(* IEC 61131-3 sources: RL_MAR/experiments/results/ablation/Ablation_antlr_only_deepseek-ai_DeepSeek-V3.2_20260611_164353 (part 3) *)

(* ---- med_75.st ---- *)
TYPE
    // State enumeration for process phases
    ProcessPhase : (
        IDLE,
        HEATING,
        BREWING,
        HOP_ADDITION,
        FERMENTATION_TRANSFER,
        COMPLETE,
        FAULT
    );

    // Status enumeration for temperature and flow
    SensorStatus : (
        NORMAL,
        LOW,
        HIGH,
        FAULT
    );
END_TYPE

FUNCTION_BLOCK HomeBrewingSystem
VAR_INPUT
    // Primary process inputs
    TemperatureSensor : REAL;        (* Current temperature in °C *)
    WaterFlowSensor : REAL;         (* Current flow rate in L/min *)
    BrewingStartTime : TIME;        (* Absolute start time of brewing process *)
    BrewingDuration : TIME;         (* Total brewing duration *)

    // Control inputs
    SystemEnable : BOOL;            (* Master enable for the system *)
    EmergencyStop : BOOL;           (* Emergency stop - overrides all outputs *)

    // Calibration inputs
    TemperatureCalibrationOffset : REAL := 0.0;  (* Temperature sensor offset *)
    FlowCalibrationFactor : REAL := 1.0;         (* Flow sensor calibration factor *)

    // Configuration inputs
    TemperatureSetpoint : REAL := 65.0;          (* Target brewing temperature *)
    TemperatureDeadband : REAL := 0.5;           (* Hysteresis for temperature control *)
    FlowThreshold : REAL := 0.5;                 (* Flow threshold for agitation *)
    FlowDeadband : REAL := 0.1;                  (* Hysteresis for flow control *)
    HopsDispenseDelay : TIME := T#5h;            (* Time delay for hops addition *)
    FermentationDelay : TIME := T#48h;           (* Time delay for fermentation transfer *)

    // Manual overrides
    ManualHeatingOverride : BOOL;                (* Manual heating control *)
    ManualAgitationOverride : BOOL;              (* Manual agitation control *)
END_VAR

VAR_OUTPUT
    // Primary control outputs
    HeatingElement : BOOL;           (* Control signal for heating element *)
    AgitationMotor : BOOL;           (* Control signal for agitation motor *)
    HopsDispenser : BOOL;            (* Control signal for hops dispenser *)
    FermentationTank : BOOL;         (* Control signal for fermentation tank transfer *)

    // Status outputs
    SystemStatus : INT;              (* Overall system status *)
    TemperatureStatus : INT;         (* Temperature sensor status *)
    FlowStatus : INT;                (* Flow sensor status *)
    ProcessPhase : INT;              (* Current process phase *)

    // Diagnostic outputs
    TemperatureAlarm : BOOL;         (* Temperature out of range alarm *)
    FlowAlarm : BOOL;                (* Flow out of range alarm *)
    BrewingElapsedTime : TIME;       (* Elapsed brewing time *)
END_VAR

VAR
    // Internal state variables
    BrewingActive : BOOL;            (* Flag indicating brewing is active *)
    HopsDispensedFlag : BOOL;        (* Flag indicating hops have been dispensed *)
    FermentationInitiatedFlag : BOOL; (* Flag indicating transfer has been initiated *)

    // Timing variables
    CurrentSystemTime : TIME;        (* Current system time *)
    BrewingElapsed : TIME;           (* Elapsed brewing time *)
    HopsDispenseTimer : TON;         (* Timer for hops dispensing *)
    FermentationTimer : TON;         (* Timer for fermentation transfer *)

    // Process variables
    TemperatureFiltered : REAL;      (* Filtered temperature reading *)
    FlowFiltered : REAL;             (* Filtered flow reading *)
    TemperatureSetpointInternal : REAL;  (* Internal setpoint with calibration *)
    FlowThresholdInternal : REAL;    (* Internal threshold with calibration *)

    // Safety and fault detection
    TemperatureSensorFault : BOOL;   (* Temperature sensor fault flag *)
    FlowSensorFault : BOOL;          (* Flow sensor fault flag *)
    SafetyInterlock : BOOL;          (* Safety interlock status *)

    // Process state
    CurrentPhase : ProcessPhase;     (* Current process phase *)

    // Configuration constants
    MIN_TEMPERATURE : REAL := 0.0;   (* Minimum valid temperature *)
    MAX_TEMPERATURE : REAL := 100.0; (* Maximum valid temperature *)
    MIN_FLOW : REAL := 0.0;          (* Minimum valid flow *)
    MAX_FLOW : REAL := 10.0;         (* Maximum valid flow *)

    // Filter constants
    TEMP_FILTER_FACTOR : REAL := 0.1;    (* Temperature filter factor *)
    FLOW_FILTER_FACTOR : REAL := 0.1;    (* Flow filter factor *)
END_VAR

// Main logic body
VAR_TEMP
    TempElapsedTime : TIME;
    TempHeatingRequired : BOOL;
    TempAgitationRequired : BOOL;
    TempHopsDispenseRequired : BOOL;
    TempFermentationRequired : BOOL;
END_VAR

// 1. Initialize and update system time
CurrentSystemTime := TIME();  // Get current system time

// 2. Apply calibration to sensor readings
TemperatureSetpointInternal := TemperatureSetpoint + TemperatureCalibrationOffset;
FlowThresholdInternal := FlowThreshold * FlowCalibrationFactor;

// 3. Apply simple low-pass filtering to sensor readings
TemperatureFiltered := TemperatureFiltered + TEMP_FILTER_FACTOR *
                      (TemperatureSensor - TemperatureFiltered);
FlowFiltered := FlowFiltered + FLOW_FILTER_FACTOR *
               (WaterFlowSensor - FlowFiltered);

// 4. Sensor validation and fault detection
TemperatureSensorFault := (TemperatureFiltered < MIN_TEMPERATURE) OR
                         (TemperatureFiltered > MAX_TEMPERATURE);
FlowSensorFault := (FlowFiltered < MIN_FLOW) OR
                  (FlowFiltered > MAX_FLOW);

// 5. Determine sensor status
IF TemperatureSensorFault THEN
    TemperatureStatus := SensorStatus.FAULT;
ELSIF TemperatureFiltered < (TemperatureSetpointInternal - 10.0) THEN
    TemperatureStatus := SensorStatus.LOW;
ELSIF TemperatureFiltered > (TemperatureSetpointInternal + 10.0) THEN
    TemperatureStatus := SensorStatus.HIGH;
ELSE
    TemperatureStatus := SensorStatus.NORMAL;
END_IF;

IF FlowSensorFault THEN
    FlowStatus := SensorStatus.FAULT;
ELSIF FlowFiltered < (FlowThresholdInternal - 0.2) THEN
    FlowStatus := SensorStatus.LOW;
ELSIF FlowFiltered > (FlowThresholdInternal + 2.0) THEN
    FlowStatus := SensorStatus.HIGH;
ELSE
    FlowStatus := SensorStatus.NORMAL;
END_IF;

// 6. Calculate elapsed brewing time
IF BrewingStartTime > T#0s THEN
    TempElapsedTime := CurrentSystemTime - BrewingStartTime;

    // Ensure elapsed time doesn't exceed duration
    IF TempElapsedTime > BrewingDuration THEN
        BrewingElapsed := BrewingDuration;
    ELSE
        BrewingElapsed := TempElapsedTime;
    END_IF;
ELSE
    BrewingElapsed := T#0s;
END_IF;

BrewingElapsedTime := BrewingElapsed;  // Output elapsed time

// 7. Determine if brewing is active
BrewingActive := (BrewingStartTime > T#0s) AND
                (BrewingElapsed < BrewingDuration) AND
                NOT EmergencyStop AND
                SystemEnable;

// 8. Process phase determination
IF EmergencyStop THEN
    CurrentPhase := ProcessPhase.FAULT;
ELSIF NOT SystemEnable THEN
    CurrentPhase := ProcessPhase.IDLE;
ELSIF NOT BrewingActive THEN
    IF BrewingElapsed >= BrewingDuration THEN
        CurrentPhase := ProcessPhase.COMPLETE;
    ELSE
        CurrentPhase := ProcessPhase.IDLE;
    END_IF;
ELSE
    // Determine phase based on elapsed time
    IF BrewingElapsed >= FermentationDelay THEN
        CurrentPhase := ProcessPhase.FERMENTATION_TRANSFER;
    ELSIF BrewingElapsed >= HopsDispenseDelay THEN
        CurrentPhase := ProcessPhase.HOP_ADDITION;
    ELSIF TemperatureFiltered >= (TemperatureSetpointInternal - TemperatureDeadband) THEN
        CurrentPhase := ProcessPhase.BREWING;
    ELSE
        CurrentPhase := ProcessPhase.HEATING;
    END_IF;
END_IF;

ProcessPhase := CurrentPhase;  // Output current phase

// 9. Heating element control with hysteresis
TempHeatingRequired := FALSE;

IF BrewingActive AND NOT TemperatureSensorFault THEN
    IF ManualHeatingOverride THEN
        TempHeatingRequired := TRUE;
    ELSIF TemperatureFiltered < (TemperatureSetpointInternal - TemperatureDeadband) THEN
        TempHeatingRequired := TRUE;
    ELSIF TemperatureFiltered >= TemperatureSetpointInternal THEN
        TempHeatingRequired := FALSE;
    END_IF;
END_IF;

HeatingElement := TempHeatingRequired AND NOT EmergencyStop;

// 10. Agitation motor control with hysteresis
TempAgitationRequired := FALSE;

IF BrewingActive AND NOT FlowSensorFault THEN
    IF ManualAgitationOverride THEN
        TempAgitationRequired := TRUE;
    ELSIF FlowFiltered > (FlowThresholdInternal + FlowDeadband) THEN
        TempAgitationRequired := TRUE;
    ELSIF FlowFiltered <= (FlowThresholdInternal - FlowDeadband) THEN
        TempAgitationRequired := FALSE;
    END_IF;
END_IF;

AgitationMotor := TempAgitationRequired AND NOT EmergencyStop;

// 11. Hops dispenser control
TempHopsDispenseRequired := FALSE;

IF BrewingActive AND (CurrentPhase = ProcessPhase.HOP_ADDITION) THEN
    // Use timer to ensure proper dispensing duration
    HopsDispenseTimer(
        IN := NOT HopsDispensedFlag,
        PT := T#10s,  // Dispense for 10 seconds
        Q => TempHopsDispenseRequired
    );

    IF HopsDispenseTimer.Q THEN
        HopsDispensedFlag := TRUE;
    END_IF;
ELSE
    HopsDispenseTimer(IN := FALSE);
END_IF;

HopsDispenser := TempHopsDispenseRequired AND NOT EmergencyStop;

// 12. Fermentation tank control
TempFermentationRequired := FALSE;

IF BrewingActive AND (CurrentPhase = ProcessPhase.FERMENTATION_TRANSFER) THEN
    // Use timer to ensure proper transfer duration
    FermentationTimer(
        IN := NOT FermentationInitiatedFlag,
        PT := T#30s,  // Transfer for 30 seconds
        Q => TempFermentationRequired
    );

    IF FermentationTimer.Q THEN
        FermentationInitiatedFlag := TRUE;
    END_IF;
ELSE
    FermentationTimer(IN := FALSE);
END_IF;

FermentationTank := TempFermentationRequired AND NOT EmergencyStop;

// 13. Alarm generation
TemperatureAlarm := (TemperatureStatus = SensorStatus.FAULT) OR
                   (TemperatureStatus = SensorStatus.HIGH) OR
                   (TemperatureStatus = SensorStatus.LOW);
FlowAlarm := (FlowStatus = SensorStatus.FAULT) OR
            (FlowStatus = SensorStatus.HIGH) OR
            (FlowStatus = SensorStatus.LOW);

// 14. System status output
IF EmergencyStop THEN
    SystemStatus := -1;  // Emergency stop active
ELSIF TemperatureSensorFault OR FlowSensorFault THEN
    SystemStatus := -2;  // Sensor fault
ELSIF NOT SystemEnable THEN
    SystemStatus := 0;   // System disabled
ELSIF CurrentPhase = ProcessPhase.IDLE THEN
    SystemStatus := 1;   // System idle
ELSIF CurrentPhase = ProcessPhase.HEATING THEN
    SystemStatus := 2;   // Heating phase
ELSIF CurrentPhase = ProcessPhase.BREWING THEN
    SystemStatus := 3;   // Brewing phase
ELSIF CurrentPhase = ProcessPhase.HOP_ADDITION THEN
    SystemStatus := 4;   // Hop addition phase
ELSIF CurrentPhase = ProcessPhase.FERMENTATION_TRANSFER THEN
    SystemStatus := 5;   // Fermentation transfer phase
ELSIF CurrentPhase = ProcessPhase.COMPLETE THEN
    SystemStatus := 6;   // Process complete
ELSE
    SystemStatus := 99;  // Unknown state
END_IF;

// 15. Reset flags when brewing is not active
IF NOT BrewingActive THEN
    HopsDispensedFlag := FALSE;
    FermentationInitiatedFlag := FALSE;
END_IF;

END_FUNCTION_BLOCK;

(* ---- med_76.st ---- *)
TYPE
    E_InstallationState : (
        STATE_IDLE,
        STATE_ACTIVE,
        STATE_SAFETY_FAULT
    );
END_TYPE

FUNCTION_BLOCK MultimediaArtInstallationControl
VAR_INPUT
    MotionSensor : BOOL; (* Motion detection input *)
    AudioTrack : BOOL; (* Selected audio track *)
    VisualContent : BOOL; (* Selected visual content *)
    SystemHealthCheck : BOOL := TRUE; (* External system health monitoring *)
    MaxActivationTime : INT := 300; (* Configurable maximum activation time *)
END_VAR

VAR_OUTPUT
    LightingControl : BOOL; (* Lighting control output *)
    AudioControl : BOOL; (* Audio playback control *)
    VisualControl : BOOL; (* Visual display control *)
    ActivationTimer : INT; (* Current activation duration *)
    CurrentState : E_InstallationState; (* For monitoring/debugging *)
    SafetyFault : BOOL; (* Indicates safety violation *)
END_VAR

VAR
    eCurrentState : E_InstallationState := STATE_IDLE;
    eNextState : E_InstallationState := STATE_IDLE;
    bInternalSafetyOK : BOOL := TRUE;
    bPowerMonitorOK : BOOL := TRUE;
END_VAR

(* Main State Machine Execution *)
CASE eCurrentState OF
    STATE_IDLE:
        (* Deactivate all multimedia elements *)
        LightingControl := FALSE;
        AudioControl := FALSE;
        VisualControl := FALSE;
        ActivationTimer := 0;
        SafetyFault := FALSE;

        (* Perform safety checks *)
        bInternalSafetyOK := SystemHealthCheck AND bPowerMonitorOK;

        (* Transition logic *)
        IF MotionSensor AND bInternalSafetyOK THEN
            eNextState := STATE_ACTIVE;
        ELSIF NOT bInternalSafetyOK THEN
            eNextState := STATE_SAFETY_FAULT;
        ELSE
            eNextState := STATE_IDLE;
        END_IF;

    STATE_ACTIVE:
        (* Activate all multimedia elements *)
        LightingControl := TRUE;
        AudioControl := AudioTrack;
        VisualControl := VisualContent;

        (* Safety Protocol: Verify all elements are properly enabled before incrementing timer *)
        IF LightingControl AND AudioControl AND VisualControl AND bInternalSafetyOK THEN
            IF ActivationTimer < MaxActivationTime THEN
                ActivationTimer := ActivationTimer + 1;
            END_IF;
        END_IF;

        (* Perform continuous safety monitoring *)
        bInternalSafetyOK := SystemHealthCheck AND bPowerMonitorOK;

        (* Transition Conditions *)
        IF NOT MotionSensor THEN
            eNextState := STATE_IDLE;
        ELSIF ActivationTimer >= MaxActivationTime THEN
            eNextState := STATE_IDLE;
        ELSIF NOT bInternalSafetyOK THEN
            eNextState := STATE_SAFETY_FAULT;
        ELSE
            eNextState := STATE_ACTIVE;
        END_IF;

    STATE_SAFETY_FAULT:
        (* Safety Protocol: Graceful shutdown *)
        LightingControl := FALSE;
        AudioControl := FALSE;
        VisualControl := FALSE;
        SafetyFault := TRUE;

        (* Monitor for safety condition resolution *)
        bInternalSafetyOK := SystemHealthCheck AND bPowerMonitorOK;

        (* Only exit safety fault when conditions are safe AND no motion detected *)
        IF bInternalSafetyOK AND NOT MotionSensor THEN
            eNextState := STATE_IDLE;
        ELSE
            eNextState := STATE_SAFETY_FAULT;
        END_IF;

END_CASE;

(* State Update *)
eCurrentState := eNextState;
CurrentState := eCurrentState;

(* Safety Protocol: Power Monitoring Simulation *)
(* This would typically interface with actual hardware monitoring *)
IF LightingControl AND AudioControl AND VisualControl THEN
    (* Simulate power load check - prevent activation if load is too high *)
    bPowerMonitorOK := TRUE; (* Replace with actual power monitoring logic *)
ELSE
    bPowerMonitorOK := TRUE;
END_IF;

END_FUNCTION_BLOCK

(* ---- med_77.st ---- *)
FUNCTION_BLOCK OutdoorLEDLightingControl
VAR_INPUT
    AmbientLight : REAL;    (* Ambient light sensor input in Lux *)
    MotionSensor : BOOL;    (* Motion sensor input (TRUE = Motion detected) *)
    EnergySaving : BOOL;    (* Energy-saving mode switch (TRUE = Energy saving ON) *)
END_VAR

VAR_OUTPUT
    Light : BOOL;           (* LED lighting control output (TRUE = Lights ON) *)
    EnergyMode : BOOL;      (* Energy-saving mode status output *)
END_VAR

VAR
    (* No internal variables required for this implementation *)
END_VAR

BEGIN
    (* Energy Mode Status: Always reflect the EnergySaving input *)
    EnergyMode := EnergySaving;

    (* Motion Detection Override - Highest Priority *)
    IF MotionSensor THEN
        Light := TRUE;      (* Override: Lights ON when motion detected *)
    ELSE
        (* Ambient Light and Energy Saving Control (when no motion detected) *)
        IF (AmbientLight < 50.0) AND (NOT EnergySaving) THEN
            Light := TRUE;  (* Lights ON: Low ambient light AND energy-saving OFF *)
        ELSE
            Light := FALSE; (* Lights OFF: Either sufficient light OR energy-saving ON *)
        END_IF;
    END_IF;
END_FUNCTION_BLOCK

(* ---- med_78.st ---- *)
(*
    FUNCTION_BLOCK: RetractableRoofControl
    DESCRIPTION: Controls a motorized retractable roof based on weather conditions.
    PRIORITY LOGIC:
        1. Combined Rain & Wind (Highest Priority): Close roof immediately.
        2. Rain Only: Close roof.
        3. Low Temperature (< 20.0°C): Close roof.
        4. Normal Conditions: Open roof.
    NOTES:
        - This is a simplified, single-output control block per the original specification.
        - The extensive I/O list and state machine from agent brQT are noted but not implemented,
          as they represent a significantly more complex system beyond the core task.
*)

FUNCTION_BLOCK RetractableRoofControl
VAR_INPUT
    RainSensor : BOOL;           (* TRUE = Rain detected *)
    WindSensor : BOOL;           (* TRUE = Strong wind detected *)
    TemperatureSensor : REAL;    (* Current ambient temperature *)
END_VAR
VAR_OUTPUT
    RoofMotor : BOOL;            (* TRUE = Close roof, FALSE = Open roof *)
END_VAR
VAR
    fTempThreshold : REAL := 20.0; (* Configurable temperature threshold *)
END_VAR

    (* Evaluate conditions in strict priority order *)
    IF (RainSensor AND WindSensor) THEN
        (* Priority 1: Combined Rain and Wind *)
        RoofMotor := TRUE;
    ELSIF (RainSensor) THEN
        (* Priority 2: Rain Only *)
        RoofMotor := TRUE;
    ELSIF (TemperatureSensor < fTempThreshold) THEN
        (* Priority 3: Low Temperature *)
        RoofMotor := TRUE;
    ELSE
        (* Priority 4: Normal Conditions *)
        RoofMotor := FALSE;
    END_IF;

END_FUNCTION_BLOCK;

(* ---- med_79.st ---- *)
(*
    CAPSULE FILLING MACHINE CONTROL FUNCTION BLOCK
    IEC 61131-3 Structured Text
    Implements a state machine with PID control for precise pharmaceutical filling
*)

TYPE E_ErrorCodes :
(
    ERR_NONE := 0,
    ERR_HOPPER_EMPTY := 1,
    ERR_OVERWEIGHT_INITIAL := 2,
    ERR_CAPSULE_DETECT_TIMEOUT := 3,
    ERR_FILLING_TIMEOUT := 4,
    ERR_EMERGENCY_STOP := 5,
    ERR_TARGET_ZERO := 6
);
END_TYPE

TYPE E_States :
(
    STATE_IDLE := 0,
    STATE_CONVEYING_IN := 1,
    STATE_FILLING := 2,
    STATE_CONVEYING_OUT := 3,
    STATE_ERROR := 99
);
END_TYPE

FUNCTION_BLOCK CapsuleFillingMachineControl
VAR_INPUT
    (* Core Process Inputs *)
    CapsuleWeight : REAL;           (* Current capsule weight measurement *)
    TargetWeight : REAL;            (* Target weight to achieve *)
    CapsuleInPosition : BOOL;       (* Capsule position sensor at entry *)
    HopperEmpty : BOOL;             (* Hopper empty sensor *)

    (* Extended Process Inputs *)
    HopperLowLevel : BOOL;          (* Hopper low level warning sensor *)
    EmergencyStop : BOOL;           (* Emergency stop button *)

    (* Timing Parameters *)
    ConveyorTime : TIME := T#2S;    (* Time to convey capsule to filling station *)
    FillingTimeout : TIME := T#10S; (* Maximum allowed filling time *)
    DetectionTimeout : TIME := T#5S;(* Timeout for capsule detection *)
    ConveyOutTime : TIME := T#2S;   (* Time to convey filled capsule out *)

    (* Control Parameters *)
    Tolerance : REAL := 0.01;       (* Weight tolerance for filling completion *)
    Kp : REAL := 1.0;               (* PID Proportional gain *)
    Ki : REAL := 0.1;               (* PID Integral gain *)
    Kd : REAL := 0.01;              (* PID Derivative gain *)
    ManualOverride : BOOL := FALSE; (* Manual override flag *)
END_VAR

VAR_OUTPUT
    (* Motor Controls *)
    FeederMotor : BOOL;             (* Controls material supply to hopper *)
    FillingMotor : BOOL;            (* Controls filling mechanism *)
    ConveyorMotor : BOOL;           (* Controls capsule conveyor *)

    (* Status Indicators *)
    FillingInProgress : BOOL;       (* TRUE during active filling *)
    WarningLight : BOOL;            (* Activated for hopper low level *)
    ErrorCode : E_ErrorCodes;       (* Current error state *)

    (* Diagnostic Outputs *)
    PIDOutput : REAL;               (* Current PID controller output *)
    WeightDeviation : REAL;         (* Deviation from target weight *)
    CurrentState : E_States;        (* Current state machine state *)
END_VAR

VAR
    (* State Machine *)
    State : E_States := STATE_IDLE;
    PreviousState : E_States;

    (* Timers *)
    ConveyorTimer : TON;
    FillingTimer : TON;
    DetectionTimer : TON;
    ConveyOutTimer : TON;

    (* PID Controller *)
    PID_Controller : PID;
    ControlOutput : REAL;
    Setpoint : REAL;
    ProcessValue : REAL;

    (* Flags *)
    CapsuleDetected : BOOL;
    WeightReached : BOOL;
    FillingComplete : BOOL;
    ConveyingComplete : BOOL;

    (* Error Handling *)
    CapsuleDetectFlag : BOOL;
    FillingTimeoutFlag : BOOL;
    OverweightError : BOOL;
    HopperLowWarning : BOOL;
    EmergencyStopActive : BOOL;

    (* Cycle Management *)
    CycleCounter : DINT;
    ErrorCounter : DINT;

    (* Weight Statistics *)
    WeightArray : ARRAY[1..100] OF REAL;
    AverageWeight : REAL;
    WeightSum : REAL := 0;
    ArrayIndex : INT := 1;
END_VAR

(* Initialize outputs *)
FeederMotor := FALSE;
FillingMotor := FALSE;
ConveyorMotor := FALSE;
FillingInProgress := FALSE;
WarningLight := FALSE;
ErrorCode := ERR_NONE;
PIDOutput := 0.0;
WeightDeviation := 0.0;
CurrentState := State;

(* Emergency Stop - Highest Priority *)
IF EmergencyStop THEN
    EmergencyStopActive := TRUE;
    ErrorCode := ERR_EMERGENCY_STOP;
    State := STATE_ERROR;
    FeederMotor := FALSE;
    FillingMotor := FALSE;
    ConveyorMotor := FALSE;
    FillingInProgress := FALSE;
    RETURN;
ELSE
    EmergencyStopActive := FALSE;
END_IF

(* Safety Check 1: Hopper Empty *)
IF HopperEmpty THEN
    ErrorCode := ERR_HOPPER_EMPTY;
    State := STATE_IDLE;
    FeederMotor := FALSE;
    FillingMotor := FALSE;
    ConveyorMotor := FALSE;
    FillingInProgress := FALSE;
    RETURN;
END_IF

(* Safety Check 2: Invalid Target Weight *)
IF TargetWeight <= 0 THEN
    ErrorCode := ERR_TARGET_ZERO;
    State := STATE_IDLE;
    FeederMotor := FALSE;
    FillingMotor := FALSE;
    ConveyorMotor := FALSE;
    FillingInProgress := FALSE;
    RETURN;
END_IF

(* Hopper Low Level Warning *)
IF HopperLowLevel THEN
    WarningLight := TRUE;
    HopperLowWarning := TRUE;
ELSE
    WarningLight := FALSE;
    HopperLowWarning := FALSE;
END_IF

(* Feeder Motor Control - runs when hopper is not empty and not in error *)
FeederMotor := NOT HopperEmpty AND NOT EmergencyStopActive;

(* Main State Machine *)
CASE State OF
    STATE_IDLE:
        (* Reset flags and timers *)
        FillingInProgress := FALSE;
        ConveyorTimer(IN := FALSE);
        FillingTimer(IN := FALSE);
        DetectionTimer(IN := FALSE);
        ConveyOutTimer(IN := FALSE);
        CapsuleDetected := FALSE;
        WeightReached := FALSE;
        FillingComplete := FALSE;
        ConveyingComplete := FALSE;

        (* Safety Check 3: Initial Overweight Detection *)
        IF CapsuleWeight >= TargetWeight THEN
            OverweightError := TRUE;
            ErrorCode := ERR_OVERWEIGHT_INITIAL;
            State := STATE_ERROR;
            RETURN;
        END_IF;

        (* Wait for capsule detection *)
        IF CapsuleInPosition THEN
            State := STATE_CONVEYING_IN;
            ConveyorTimer(IN := TRUE, PT := ConveyorTime);
            DetectionTimer(IN := TRUE, PT := DetectionTimeout);
        END_IF;

    STATE_CONVEYING_IN:
        (* Activate conveyor to move capsule to filling station *)
        ConveyorMotor := TRUE;
        ConveyorTimer(IN := TRUE);
        DetectionTimer(IN := TRUE);

        (* Check for successful conveyance *)
        IF ConveyorTimer.Q THEN
            ConveyingComplete := TRUE;
            ConveyorTimer(IN := FALSE);
            DetectionTimer(IN := FALSE);
            State := STATE_FILLING;
            FillingTimer(IN := TRUE, PT := FillingTimeout);

        (* Check for capsule detection timeout *)
        ELSIF DetectionTimer.Q THEN
            CapsuleDetectFlag := TRUE;
            ErrorCode := ERR_CAPSULE_DETECT_TIMEOUT;
            ConveyorTimer(IN := FALSE);
            DetectionTimer(IN := FALSE);
            State := STATE_ERROR;
        END_IF;

    STATE_FILLING:
        (* Set filling status *)
        FillingInProgress := TRUE;

        (* Configure PID Controller *)
        Setpoint := TargetWeight;
        ProcessValue := CapsuleWeight;

        (* Initialize PID parameters on first entry *)
        IF PreviousState <> STATE_FILLING THEN
            PID_Controller.Kp := Kp;
            PID_Controller.Ki := Ki;
            PID_Controller.Kd := Kd;
            PID_Controller.Ts := T#20MS;  (* Sample time *)
        END_IF;

        (* Execute PID control *)
        PID_Controller(
            Setpoint := Setpoint,
            ProcessValue := ProcessValue,
            ControlOutput => ControlOutput
        );

        (* Convert PID output to motor control *)
        PIDOutput := ControlOutput;
        IF ControlOutput > 0.0 AND CapsuleWeight < (TargetWeight - Tolerance) THEN
            FillingMotor := TRUE;
        ELSE
            FillingMotor := FALSE;
        END_IF;

        (* Monitor filling progress *)
        FillingTimer(IN := TRUE);
        WeightDeviation := TargetWeight - CapsuleWeight;

        (* Check for successful filling completion *)
        IF CapsuleWeight >= (TargetWeight - Tolerance) AND CapsuleWeight <= (TargetWeight + Tolerance) THEN
            WeightReached := TRUE;
            FillingMotor := FALSE;
            FillingTimer(IN := FALSE);
            FillingComplete := TRUE;

            (* Record weight for statistics *)
            WeightArray[ArrayIndex] := CapsuleWeight;
            WeightSum := WeightSum + CapsuleWeight;
            ArrayIndex := ArrayIndex MOD 100 + 1;

            (* Calculate average weight *)
            AverageWeight := WeightSum / CycleCounter;

            State := STATE_CONVEYING_OUT;
            ConveyOutTimer(IN := TRUE, PT := ConveyOutTime);

        (* Check for filling timeout *)
        ELSIF FillingTimer.Q THEN
            FillingTimeoutFlag := TRUE;
            ErrorCode := ERR_FILLING_TIMEOUT;
            FillingMotor := FALSE;
            FillingTimer(IN := FALSE);
            State := STATE_ERROR;
        END_IF;

    STATE_CONVEYING_OUT:
        (* Activate conveyor to move filled capsule out *)
        ConveyorMotor := TRUE;
        ConveyOutTimer(IN := TRUE);

        IF ConveyOutTimer.Q THEN
            ConveyorMotor := FALSE;
            ConveyOutTimer(IN := FALSE);
            FillingInProgress := FALSE;
            CycleCounter := CycleCounter + 1;
            State := STATE_IDLE;
        END_IF;

    STATE_ERROR:
        (* Error State - All motors off *)
        FeederMotor := FALSE;
        FillingMotor := FALSE;
        ConveyorMotor := FALSE;
        FillingInProgress := FALSE;

        (* Reset error on manual intervention or condition change *)
        IF NOT EmergencyStopActive AND
           NOT HopperEmpty AND
           CapsuleWeight < TargetWeight AND
           CapsuleInPosition THEN
            ErrorCode := ERR_NONE;
            CapsuleDetectFlag := FALSE;
            FillingTimeoutFlag := FALSE;
            OverweightError := FALSE;
            ErrorCounter := ErrorCounter + 1;
            State := STATE_IDLE;
        END_IF;

END_CASE;

(* Store previous state for edge detection *)
PreviousState := State;

END_FUNCTION_BLOCK

(* ---- med_80.st ---- *)
FUNCTION_BLOCK DoughMixerControl
VAR_INPUT
    IngredientsDetected : BOOL;
END_VAR

VAR_OUTPUT
    MixingInProgress : BOOL;
END_VAR

VAR
    MixingTimeElapsed : TIME;
    MixingTimeLimit : TIME := T#5S;
    PrevIngredientsDetected : BOOL;
END_VAR

(* Rising edge detection for ingredient presence *)
IF NOT PrevIngredientsDetected AND IngredientsDetected THEN
    MixingInProgress := TRUE;
    MixingTimeElapsed := T#0S;
END_IF;

(* Stop conditions: ingredients removed OR time limit reached *)
IF NOT IngredientsDetected OR (MixingTimeElapsed >= MixingTimeLimit) THEN
    MixingInProgress := FALSE;
END_IF;

(* Timer increment only while mixing is active *)
IF MixingInProgress THEN
    MixingTimeElapsed := MixingTimeElapsed + T#1S;
END_IF;

(* Store previous state for edge detection *)
PrevIngredientsDetected := IngredientsDetected;

END_FUNCTION_BLOCK;

(* ---- med_81.st ---- *)
FUNCTION_BLOCK SolarPanelTracking
VAR_INPUT
    CurrentTime : TIME;
    SolarIntensity : REAL;
END_VAR

VAR_OUTPUT
    PanelAngle : REAL;
END_VAR

VAR
    SunriseTime : TIME := T#6H;
    NoonTime : TIME := T#12H;
    SunsetTime : TIME := T#18H;
    MorningAngle : REAL := 30.0;
    NoonAngle : REAL := 60.0;
    EveningAngle : REAL := 30.0;
END_VAR

(* Solar intensity override takes precedence *)
IF SolarIntensity >= 90.0 THEN
    PanelAngle := NoonAngle;
ELSE
    (* Time-based tracking logic *)
    IF (CurrentTime < SunriseTime) OR (CurrentTime >= SunsetTime) THEN
        PanelAngle := 0.0; (* Nighttime - panel horizontal *)
    ELSIF (CurrentTime >= SunriseTime) AND (CurrentTime < NoonTime) THEN
        PanelAngle := MorningAngle; (* Morning period *)
    ELSIF (CurrentTime >= NoonTime) AND (CurrentTime < SunsetTime) THEN
        PanelAngle := EveningAngle; (* Afternoon/Evening period *)
    ELSE
        PanelAngle := 0.0; (* Fallback safety position *)
    END_IF;
END_IF;

END_FUNCTION_BLOCK;

(* ---- med_82.st ---- *)
FUNCTION_BLOCK PetFeederControl
VAR_INPUT
    CurrentTime : TIME; (* Current system time from RTC *)
END_VAR

VAR_OUTPUT
    FoodDispense : BOOL; (* Food dispenser control signal *)
END_VAR

VAR
    FeedTime1 : TIME := T#8H0M0S; (* First feeding time - 8:00 AM *)
    FeedTime2 : TIME := T#12H0M0S; (* Second feeding time - 12:00 PM *)
    FeedTime3 : TIME := T#18H0M0S; (* Third feeding time - 6:00 PM *)
    FoodAmount : INT := 50; (* Amount of food to dispense in grams - Currently unused *)
END_VAR

(* Main dispensing logic *)
FoodDispense := (CurrentTime >= FeedTime1) AND (CurrentTime < FeedTime1 + T#30S)
             OR (CurrentTime >= FeedTime2) AND (CurrentTime < FeedTime2 + T#30S)
             OR (CurrentTime >= FeedTime3) AND (CurrentTime < FeedTime3 + T#30S);

END_FUNCTION_BLOCK

(* ---- med_83.st ---- *)
(*
    FUNCTION_BLOCK AmusementRideControl
    Safety control system for an amusement ride with strict fail-safe principles.

    Safety Properties Verified:
    1. Emergency Stop has highest priority and immediately stops motor
    2. Motor and Brake are never active simultaneously
    3. Motor only runs when ALL start conditions are met
    4. System defaults to safe state (brake engaged, motor off)

    Inputs:
        StartButton  : BOOL  - Start command (must be TRUE to run)
        StopButton   : BOOL  - Emergency stop (TRUE = emergency active)
        SpeedSensor  : REAL  - Current speed measurement (RPM)
        SafetySensor : BOOL  - Safety interlock status (TRUE = safe)

    Outputs:
        MotorOn : BOOL - Motor control (TRUE = run, FALSE = stop)
        BrakeOn : BOOL - Brake control (TRUE = engaged, FALSE = released)

    Internal:
        SpeedLimit : REAL - Maximum allowed speed (RPM)
*)

FUNCTION_BLOCK AmusementRideControl
VAR_INPUT
    StartButton  : BOOL;  (* Start button input *)
    StopButton   : BOOL;  (* Emergency stop button input *)
    SpeedSensor  : REAL;  (* Speed sensor input (RPM) *)
    SafetySensor : BOOL;  (* Safety sensor status *)
END_VAR

VAR_OUTPUT
    MotorOn : BOOL := FALSE;  (* Motor control output *)
    BrakeOn : BOOL := TRUE;   (* Brake control output - Default to safe state *)
END_VAR

VAR
    SpeedLimit : REAL := 60.0;  (* Maximum allowed speed in RPM *)
END_VAR

(* Main Safety Logic *)
METHOD SafetyLogic : BOOL
VAR_INPUT
    bStartReq    : BOOL;
    bEmergency   : BOOL;
    rCurrentSpeed : REAL;
    rSpeedLimit   : REAL;
    bSafetyOK    : BOOL;
END_VAR
VAR_OUTPUT
    bMotorPermit : BOOL;
END_VAR
    (* Emergency Stop has ABSOLUTE highest priority *)
    IF bEmergency THEN
        bMotorPermit := FALSE;
        RETURN;
    END_IF;

    (* All start conditions must be met simultaneously *)
    bMotorPermit := bStartReq
                    AND (rCurrentSpeed <= rSpeedLimit)
                    AND bSafetyOK;
END_METHOD

(* Main execution body *)
METHOD Execute
    LOCAL_VAR
        bSafeToRun : BOOL;
    END_VAR

    (* Determine if it's safe to run the motor *)
    SafetyLogic(
        bStartReq := StartButton,
        bEmergency := StopButton,
        rCurrentSpeed := SpeedSensor,
        rSpeedLimit := SpeedLimit,
        bSafetyOK := SafetySensor,
        bMotorPermit => bSafeToRun
    );

    (* Apply safety logic with emergency stop override *)
    IF StopButton THEN
        (* CRITICAL: Emergency Stop - Highest Priority *)
        MotorOn := FALSE;
        BrakeOn := TRUE;
    ELSE
        (* Normal operation based on safety logic *)
        MotorOn := bSafeToRun;
        BrakeOn := NOT bSafeToRun;  (* Brake is opposite of motor state *)
    END_IF;

    (* Final safety assertion: Ensure brake is engaged if motor is off *)
    IF NOT MotorOn THEN
        BrakeOn := TRUE;
    END_IF;
END_METHOD

(* Initialization method *)
METHOD Init
    (* Initialize outputs to safe state *)
    MotorOn := FALSE;
    BrakeOn := TRUE;

    (* Initialize speed limit *)
    SpeedLimit := 60.0;
END_METHOD

END_FUNCTION_BLOCK;

(* ---- med_84.st ---- *)
(* ============================================================================
   FUNCTION_BLOCK: ParcelSortingSystem
   Description: Implements control logic for a parcel sorting system.
                Routes parcels based on size and destination code.
   Inputs:  ParcelSizeSensor (REAL), DestinationCodeSensor (INT)
   Outputs: ConveyorBeltMotor (BOOL), SortingGate1 (BOOL), SortingGate2 (BOOL)
   Safety: Invalid inputs stop the conveyor and close all gates.
   Author: Senior PLC Commissioning Engineer
   Standard: IEC 61131-3
   ============================================================================ *)

FUNCTION_BLOCK ParcelSortingSystem
VAR_INPUT
    ParcelSizeSensor : REAL;     (* Measured parcel size [units] *)
    DestinationCodeSensor : INT; (* Destination code: 1=Location A, 2=Location B *)
END_VAR

VAR_OUTPUT
    ConveyorBeltMotor : BOOL; (* TRUE = Motor ON / Conveyor moving *)
    SortingGate1      : BOOL; (* TRUE = Gate 1 OPEN (for large parcels) *)
    SortingGate2      : BOOL; (* TRUE = Gate 2 OPEN (for small to Location A) *)
END_VAR

VAR
    (* Internal Constants *)
    SizeThreshold : REAL := 50.0;   (* Threshold to distinguish large vs. small parcels *)
    MinValidSize  : REAL := 0.01;   (* Minimum valid size to reject zero/negative values *)
    MaxValidSize  : REAL := 1000.0; (* Maximum valid size for sensor range *)
    DestCodeA     : INT := 1;       (* Destination code for Location A *)
    DestCodeB     : INT := 2;       (* Destination code for Location B *)

    (* Internal Flags *)
    bSizeValid    : BOOL; (* TRUE if ParcelSizeSensor is within valid range *)
    bDestValid    : BOOL; (* TRUE if DestinationCodeSensor is 1 or 2 *)
    bInputsValid  : BOOL; (* TRUE if both size and destination are valid *)
END_VAR

(* ============================================================================
   Main Logic Body
   ============================================================================ *)
    (* 1. Input Validation *)
    bSizeValid := (ParcelSizeSensor >= MinValidSize) AND (ParcelSizeSensor <= MaxValidSize);
    bDestValid := (DestinationCodeSensor = DestCodeA) OR (DestinationCodeSensor = DestCodeB);
    bInputsValid := bSizeValid AND bDestValid;

    (* 2. Core Sorting Logic *)
    IF bInputsValid THEN
        (* Valid inputs detected - activate conveyor *)
        ConveyorBeltMotor := TRUE;

        (* Determine parcel routing based on size and destination *)
        IF ParcelSizeSensor > SizeThreshold THEN
            (* LARGE PARCEL: Route to Gate 1, regardless of destination *)
            SortingGate1 := TRUE;
            SortingGate2 := FALSE;
        ELSE
            (* SMALL PARCEL: Route based on destination code *)
            SortingGate1 := FALSE; (* Gate 1 always closed for small parcels *)

            CASE DestinationCodeSensor OF
                DestCodeA:
                    (* Small parcel to Location A: Route to Gate 2 *)
                    SortingGate2 := TRUE;
                DestCodeB:
                    (* Small parcel to Location B: No diversion, keep on main belt *)
                    SortingGate2 := FALSE;
                ELSE
                    (* This case should not occur due to prior validation,
                       but set safe default. *)
                    SortingGate2 := FALSE;
            END_CASE;
        END_IF;
    ELSE
        (* INVALID INPUTS: Safe shutdown state *)
        ConveyorBeltMotor := FALSE;
        SortingGate1      := FALSE;
        SortingGate2      := FALSE;
    END_IF;

END_FUNCTION_BLOCK;

(* ---- med_85.st ---- *)
(*
    ShredderControl FUNCTION_BLOCK
    Final, production-ready implementation.
    Synthesized from specialist agent inputs with critical evaluation.
    Compliant with IEC 61131-3 standard.
*)

FUNCTION_BLOCK ShredderControl
VAR_INPUT
    StartButton : BOOL;        (* Momentary start command *)
    StopButton : BOOL;         (* Momentary stop command *)
    EmergencyStop : BOOL;      (* NC contact, TRUE = pressed/fault *)
    MaterialInFeed : BOOL;     (* Presence detected in feed chute *)
    JammedSensor : BOOL;       (* TRUE when a jam is detected *)
END_VAR
VAR_OUTPUT
    MotorControl : BOOL;       (* Command to motor starter *)
    SafetyRelay : BOOL;        (* Command to safety relay coil *)
END_VAR
VAR
    fbMotorLatch : SR;         (* Standard Set-Reset Latch for motor state *)
    bEmergencyCondition : BOOL;(* Consolidated emergency signal *)
    bRunPermissive : BOOL;     (* Permissive for normal run requests *)
END_VAR

(* --- Priority 1: Determine Emergency Condition --- *)
bEmergencyCondition := EmergencyStop OR JammedSensor;

(* --- Priority 2: Safety Relay Logic (Directly controlled by safety state) --- *)
SafetyRelay := NOT bEmergencyCondition;

(* --- Priority 3: Normal Run Permissive Logic --- *)
bRunPermissive := NOT bEmergencyCondition AND NOT StopButton;

(* --- Priority 4: Motor Latch Logic --- *)
(* Set Condition: Permissive is TRUE AND (Start button pressed OR material in feed) *)
fbMotorLatch(S1 := bRunPermissive AND (StartButton OR MaterialInFeed),
             R  := NOT bRunPermissive); (* Reset if permissive is lost *)

(* --- Final Motor Output Assignment --- *)
(* Motor runs only if the latch is set AND the safety relay is active (fail-safe check) *)
MotorControl := fbMotorLatch.Q1 AND SafetyRelay;

END_FUNCTION_BLOCK

(* ---- med_86.st ---- *)
FUNCTION_BLOCK FruitJuicingBottling
VAR_INPUT
    StartButton : BOOL;    (* Rising edge trigger to start the process *)
    StopButton : BOOL;     (* Level-sensitive command to stop the process *)
    FruitSelected : BOOL;  (* System readiness signal - must be TRUE to run *)
END_VAR

VAR_OUTPUT
    JuiceProcessing : BOOL;    (* Controls the juice extraction stage *)
    BottleFilling : BOOL;      (* Controls the bottle filling stage *)
    CapPlacement : BOOL;       (* Controls the cap placement stage *)
    Packaging : BOOL;          (* Controls the packaging stage *)
    ProcessInProgress : BOOL;  (* System status indicator *)
END_VAR

VAR
    bProcessActive : BOOL := FALSE;  (* Internal process state memory *)
END_VAR

(* Main Process State Machine *)
(* Start condition: Rising edge detection on StartButton with prerequisites *)
IF StartButton AND FruitSelected AND NOT bProcessActive THEN
    bProcessActive := TRUE;
END_IF;

(* Stop conditions: Level-sensitive stop commands *)
IF StopButton OR NOT FruitSelected THEN
    bProcessActive := FALSE;
END_IF;

(* Process Stage Outputs - All stages run concurrently when process is active *)
JuiceProcessing := bProcessActive;
BottleFilling := bProcessActive;
CapPlacement := bProcessActive;
Packaging := bProcessActive;

(* Process Status Output *)
ProcessInProgress := bProcessActive;

END_FUNCTION_BLOCK

(* ---- med_87.st ---- *)
FUNCTION_BLOCK WaterDesalination
VAR_INPUT
    StartButton : BOOL;        (* Input for starting the desalination process *)
    StopButton : BOOL;         (* Input for stopping the desalination process *)
    SalinitySensor : REAL;     (* Input for salinity level measurement *)
END_VAR

VAR_OUTPUT
    SeawaterInletValve : BOOL;         (* Output for seawater inlet valve control *)
    FreshwaterOutletValve : BOOL;      (* Output for freshwater outlet valve control *)
    DesalinationInProgress : BOOL;     (* Indicator for an ongoing desalination process *)
END_VAR

VAR
    MaxSalinity : REAL := 35.0;        (* Maximum allowable salinity in ppm for freshwater *)
    SalinityControlSeconds : INT := 0; (* Timer for salinity control in seconds *)
    SalinityTimer : TON;               (* IEC 61131-3 timer for 10-second intervals *)
END_VAR

(* Salinity Timer Execution *)
SalinityTimer(IN := DesalinationInProgress, PT := T#10S);

(* Process Start/Stop Control *)
IF StopButton THEN
    DesalinationInProgress := FALSE;
    SeawaterInletValve := FALSE;
    FreshwaterOutletValve := FALSE;
    SalinityControlSeconds := 0;
ELSIF StartButton AND NOT DesalinationInProgress THEN
    DesalinationInProgress := TRUE;
    SeawaterInletValve := TRUE;
    FreshwaterOutletValve := TRUE;
END_IF;

(* Salinity Monitoring and Control *)
IF SalinityTimer.Q THEN
    SalinityControlSeconds := SalinityControlSeconds + 10;

    IF DesalinationInProgress THEN
        IF SalinitySensor > MaxSalinity THEN
            FreshwaterOutletValve := FALSE;
        ELSE
            FreshwaterOutletValve := TRUE;
        END_IF;
    END_IF;
END_IF;

END_FUNCTION_BLOCK

(* ---- med_88.st ---- *)
FUNCTION_BLOCK SmartLockerControl
VAR_INPUT
    AccessCode : INT;     (* User-provided access code *)
    LockerNumber : INT;   (* Selected locker number (1-10) *)
END_VAR

VAR_OUTPUT
    LockerOpen : BOOL;    (* TRUE when access is granted and locker should open *)
END_VAR

VAR
    LockerStatus : ARRAY[1..10] OF BOOL;      (* TRUE=occupied/locked, FALSE=empty/unlocked *)
    LockerAccessCode : ARRAY[1..10] OF INT;   (* Stored access codes for each locker *)
    bInitialized : BOOL := FALSE;             (* One-time initialization flag *)
END_VAR

(* One-time initialization of locker data *)
IF NOT bInitialized THEN
    (* Initialize all lockers to locked state (TRUE) *)
    LockerStatus[1] := TRUE;
    LockerStatus[2] := TRUE;
    LockerStatus[3] := TRUE;
    LockerStatus[4] := TRUE;
    LockerStatus[5] := TRUE;
    LockerStatus[6] := TRUE;
    LockerStatus[7] := TRUE;
    LockerStatus[8] := TRUE;
    LockerStatus[9] := TRUE;
    LockerStatus[10] := TRUE;

    (* Set predefined access codes *)
    LockerAccessCode[1] := 1234;
    LockerAccessCode[2] := 5678;
    LockerAccessCode[3] := 9876;
    LockerAccessCode[4] := 4321;
    LockerAccessCode[5] := 6543;
    LockerAccessCode[6] := 7890;
    LockerAccessCode[7] := 3456;
    LockerAccessCode[8] := 8765;
    LockerAccessCode[9] := 2345;
    LockerAccessCode[10] := 6789;

    bInitialized := TRUE;
END_IF;

(* Main access control logic *)
LockerOpen := FALSE;  (* Default state - locker remains closed *)

(* Validate locker number range *)
IF (LockerNumber >= 1) AND (LockerNumber <= 10) THEN
    (* Verify access code matches stored code for specified locker *)
    IF AccessCode = LockerAccessCode[LockerNumber] THEN
        (* Grant access and update locker status *)
        LockerOpen := TRUE;
        LockerStatus[LockerNumber] := FALSE;  (* Locker becomes empty/unlocked *)
    END_IF;
END_IF;

END_FUNCTION_BLOCK

(* ---- med_89.st ---- *)
FUNCTION_BLOCK SoilTestingDeviceControl
VAR_INPUT
    StartButton : BOOL; (* Input for starting the testing process *)
    SoilSampleDetected : BOOL; (* Input for detecting soil sample *)
END_VAR
VAR_OUTPUT
    NutrientPump : BOOL; (* Output to control nutrient pump *)
    pHAdjustmentPump : BOOL; (* Output to control pH adjustment pump *)
END_VAR
VAR
    pHSensorValue : REAL; (* Simulated pH sensor value *)
    NutrientSensorValue : REAL; (* Simulated nutrient sensor value *)
    TestingStatus : INT; (* Status: 0=Idle, 1=Testing, 2=Completed *)
    NutrientThreshold : REAL := 0.7; (* Nutrient level threshold for analysis *)
    pHThreshold : REAL := 6.5; (* pH level threshold for analysis *)
END_VAR

CASE TestingStatus OF
    0: (* Idle State *)
        (* Initialize sensor values *)
        pHSensorValue := 7.0;
        NutrientSensorValue := 0.5;

        (* Ensure pumps are deactivated *)
        NutrientPump := FALSE;
        pHAdjustmentPump := FALSE;

        (* Check for start condition *)
        IF StartButton THEN
            TestingStatus := 1;
            NutrientPump := TRUE;
            pHAdjustmentPump := TRUE;
        END_IF;

    1: (* Testing State *)
        (* Update sensor values during testing *)
        NutrientSensorValue := NutrientSensorValue + 0.1;
        pHSensorValue := pHSensorValue - 0.5;

        (* Enforce sensor value boundaries *)
        IF NutrientSensorValue > 0.9 THEN
            NutrientSensorValue := 0.9;
        END_IF;

        IF pHSensorValue < 4.0 THEN
            pHSensorValue := 4.0;
        END_IF;

        (* Check for completion condition *)
        IF SoilSampleDetected THEN
            IF (NutrientSensorValue >= NutrientThreshold) AND (pHSensorValue <= pHThreshold) THEN
                TestingStatus := 2;
                NutrientPump := FALSE;
                pHAdjustmentPump := FALSE;
            END_IF;
        END_IF;

    2: (* Completed State *)
        (* Ensure pumps are deactivated *)
        NutrientPump := FALSE;
        pHAdjustmentPump := FALSE;

        (* Reset to Idle when StartButton is released *)
        IF NOT StartButton THEN
            TestingStatus := 0;
        END_IF;

END_CASE;

END_FUNCTION_BLOCK

(* ---- med_90.st ---- *)
FUNCTION_BLOCK SushiConveyorControl
VAR_INPUT
    StartButton : BOOL;    (* Input to start the conveyor *)
    StopButton : BOOL;     (* Input to stop the conveyor *)
    EmergencyStop : BOOL;  (* Input for emergency stop *)
END_VAR

VAR_OUTPUT
    ConveyorMotor : BOOL;  (* Output to control the conveyor motor *)
END_VAR

VAR
    BeltRunning : BOOL;    (* Status of the conveyor: Running or Stopped *)
    ConveyorTimer : INT;   (* Timer counter for conveyor rotation *)
    RotationTime : INT := 5; (* Time for one rotation in seconds *)
    tonTimer : TON;        (* Timer function block for precise timing *)
END_VAR

(* Initialization *)
BeltRunning := FALSE;
ConveyorTimer := 0;

(* Emergency Stop - Highest Priority *)
IF EmergencyStop THEN
    ConveyorMotor := FALSE;
    BeltRunning := FALSE;
    ConveyorTimer := 0;
    tonTimer(IN := FALSE, PT := T#0S);
    RETURN;
END_IF;

(* Start/Stop Control with priority to Stop *)
IF StopButton AND BeltRunning THEN
    ConveyorMotor := FALSE;
    BeltRunning := FALSE;
    ConveyorTimer := 0;
    tonTimer(IN := FALSE, PT := T#0S);
ELSIF StartButton AND NOT BeltRunning AND NOT StopButton THEN
    ConveyorMotor := TRUE;
    BeltRunning := TRUE;
    ConveyorTimer := 0;
    tonTimer(IN := FALSE, PT := T#0S);
END_IF;

(* Simulated Rotation - Timer-based cycle *)
IF BeltRunning THEN
    (* Use TON timer for precise timing *)
    tonTimer(IN := TRUE, PT := T#1S);

    IF tonTimer.Q THEN
        ConveyorTimer := ConveyorTimer + 1;
        tonTimer(IN := FALSE, PT := T#0S);

        (* Check if rotation time reached *)
        IF ConveyorTimer >= RotationTime THEN
            ConveyorTimer := 0;
        END_IF;
    END_IF;

    (* Keep motor running while belt is running *)
    ConveyorMotor := TRUE;
END_IF;

END_FUNCTION_BLOCK

(* ---- med_91.st ---- *)
TYPE
    AGV_Status : STRUCT
        IsReady : BOOL;
        IsWorking : BOOL;
        CurrentTask : INT; (* 0 = no task *)
        Position : INT;
    END_STRUCT;
END_TYPE

FUNCTION_BLOCK AGVControlSystem
VAR_INPUT
    MaterialRequest : INT; (* New material request, positive value indicates valid request *)
    TaskComplete : ARRAY[1..3] OF BOOL; (* External signal to indicate AGV task completion *)
END_VAR
VAR_OUTPUT
    AGV1_Ready : BOOL := TRUE;
    AGV2_Ready : BOOL := TRUE;
    AGV3_Ready : BOOL := TRUE;
    QueueCount : INT := 0; (* Current number of pending tasks *)
    SystemError : BOOL := FALSE; (* Indicates system error state *)
END_VAR
VAR
    MaterialQueue : ARRAY[1..10] OF INT; (* FIFO queue for material requests *)
    QueueHead : INT := 1; (* Index of next task to assign *)
    QueueTail : INT := 1; (* Index where next request will be stored *)

    AGVs : ARRAY[1..3] OF AGV_Status := [
        (IsReady := TRUE, IsWorking := FALSE, CurrentTask := 0, Position := 0),
        (IsReady := TRUE, IsWorking := FALSE, CurrentTask := 0, Position := 0),
        (IsReady := TRUE, IsWorking := FALSE, CurrentTask := 0, Position := 0)
    ];

    i : INT;
    TempRequest : INT;
    TaskAssigned : BOOL;
END_VAR

(* Initialize outputs *)
AGV1_Ready := AGVs[1].IsReady;
AGV2_Ready := AGVs[2].IsReady;
AGV3_Ready := AGVs[3].IsReady;
QueueCount := 0; (* Will be calculated below *)
SystemError := FALSE;

(* Calculate actual queue count *)
QueueCount := 0;
FOR i := 1 TO 10 DO
    IF MaterialQueue[i] > 0 THEN
        QueueCount := QueueCount + 1;
    END_IF;
END_FOR;

(* 1. Handle new material requests with validation *)
IF MaterialRequest > 0 THEN
    (* Check for queue overflow *)
    IF QueueCount < 10 THEN
        (* Store request in queue *)
        MaterialQueue[QueueTail] := MaterialRequest;

        (* Update queue tail with wrap-around *)
        QueueTail := QueueTail + 1;
        IF QueueTail > 10 THEN
            QueueTail := 1;
        END_IF;

        QueueCount := QueueCount + 1;
    ELSE
        (* Queue overflow error *)
        SystemError := TRUE;
    END_IF;
END_IF;

(* 2. Handle task completion signals *)
FOR i := 1 TO 3 DO
    IF TaskComplete[i] AND AGVs[i].IsWorking THEN
        (* Reset AGV status upon task completion *)
        AGVs[i].IsWorking := FALSE;
        AGVs[i].CurrentTask := 0;
        AGVs[i].IsReady := TRUE;

        (* Safety: Ensure position is non-negative *)
        IF AGVs[i].Position < 0 THEN
            AGVs[i].Position := 0;
        END_IF;
    END_IF;
END_FOR;

(* 3. Priority-based task assignment (AGV1 > AGV2 > AGV3) *)
TaskAssigned := FALSE;

(* Check AGV1 first *)
IF (QueueCount > 0) AND (NOT TaskAssigned) THEN
    IF AGVs[1].IsReady AND (NOT AGVs[1].IsWorking) THEN
        (* Assign task to AGV1 *)
        AGVs[1].CurrentTask := MaterialQueue[QueueHead];
        AGVs[1].IsWorking := TRUE;
        AGVs[1].IsReady := FALSE;

        (* Remove task from queue *)
        MaterialQueue[QueueHead] := 0;

        (* Update queue head with wrap-around *)
        QueueHead := QueueHead + 1;
        IF QueueHead > 10 THEN
            QueueHead := 1;
        END_IF;

        QueueCount := QueueCount - 1;
        TaskAssigned := TRUE;
    END_IF;
END_IF;

(* Check AGV2 if AGV1 is busy *)
IF (QueueCount > 0) AND (NOT TaskAssigned) THEN
    IF AGVs[2].IsReady AND (NOT AGVs[2].IsWorking) THEN
        (* Assign task to AGV2 *)
        AGVs[2].CurrentTask := MaterialQueue[QueueHead];
        AGVs[2].IsWorking := TRUE;
        AGVs[2].IsReady := FALSE;

        (* Remove task from queue *)
        MaterialQueue[QueueHead] := 0;

        (* Update queue head with wrap-around *)
        QueueHead := QueueHead + 1;
        IF QueueHead > 10 THEN
            QueueHead := 1;
        END_IF;

        QueueCount := QueueCount - 1;
        TaskAssigned := TRUE;
    END_IF;
END_IF;

(* Check AGV3 if AGV1 and AGV2 are busy *)
IF (QueueCount > 0) AND (NOT TaskAssigned) THEN
    IF AGVs[3].IsReady AND (NOT AGVs[3].IsWorking) THEN
        (* Assign task to AGV3 *)
        AGVs[3].CurrentTask := MaterialQueue[QueueHead];
        AGVs[3].IsWorking := TRUE;
        AGVs[3].IsReady := FALSE;

        (* Remove task from queue *)
        MaterialQueue[QueueHead] := 0;

        (* Update queue head with wrap-around *)
        QueueHead := QueueHead + 1;
        IF QueueHead > 10 THEN
            QueueHead := 1;
        END_IF;

        QueueCount := QueueCount - 1;
        TaskAssigned := TRUE;
    END_IF;
END_IF;

(* 4. Update AGV positions for working AGVs *)
FOR i := 1 TO 3 DO
    IF AGVs[i].IsWorking THEN
        (* Simulate position update - in real system this would come from sensors *)
        AGVs[i].Position := AGVs[i].Position + 1;

        (* Safety constraint: Ensure position is non-negative *)
        IF AGVs[i].Position < 0 THEN
            AGVs[i].Position := 0;
        END_IF;
    END_IF;
END_FOR;

(* 5. Final output updates *)
AGV1_Ready := AGVs[1].IsReady;
AGV2_Ready := AGVs[2].IsReady;
AGV3_Ready := AGVs[3].IsReady;

(* 6. Additional error checking *)
(* Check for invalid queue state *)
IF (QueueCount < 0) OR (QueueCount > 10) THEN
    SystemError := TRUE;
END_IF;

(* Check for invalid AGV states *)
FOR i := 1 TO 3 DO
    IF AGVs[i].IsWorking AND AGVs[i].IsReady THEN
        SystemError := TRUE;
    END_IF;

    IF (AGVs[i].CurrentTask > 0) AND (NOT AGVs[i].IsWorking) THEN
        SystemError := TRUE;
    END_IF;
END_FOR;

END_FUNCTION_BLOCK;
